Yaskawa INFORM job: R1_W01(KAMERA)(0,-90).JBI

/JOB
//NAME R1_W01(KAMERA)(0,-90)
//POS
///NPOS 10,10,0,0,0,0
///TOOL 0
///POSTYPE PULSE
///LIMIT ON
///PULSE
C00000=3343,-162524,-138229,-10688,931,-77458
C00001=3343,-162524,-138229,-10688,931,-77458
///LIMIT OFF
C00002=146555,-32624,-97126,-37706,85917,-68564
C00003=192498,68076,-33610,-32500,114040,-68788
C00004=185826,59216,-21978,-23322,112796,-65701
C00005=180860,70259,-8687,-21392,109491,-66464
C00006=183450,60909,-15972,-26835,103470,-66374
C00007=180988,72118,-8747,-21583,110442,-66611
C00008=181141,75755,-9105,-21978,112418,-66957
C00009=188486,40732,-78117,-36575,78939,-72193
BC00000=7717,939738,1042121
BC00001=7717,1361376,1042121
///LIMIT ON
BC00002=130580,1376610,1059176
BC00003=195745,1384690,1068222
BC00004=189788,1384690,1068222
BC00005=189788,1384690,1068222
BC00006=189789,1384690,1068220
BC00007=189953,1384690,1068222
BC00008=189837,1384690,1068222
BC00009=229747,1383410,1068222
//INST
///DATE 2024/07/30 12:51
///ATTR SC,RW
///GROUP1 RB1,BS1
NOP
'r1_W01(kamera)(0,-90)
'Path W401
SFTOF
MOVJ C00000 BC00000 VJ=100.00
MOVJ C00001 BC00001 VJ=100.00
MOVJ C00002 BC00002 VJ=100.00
MOVJ C00003 BC00003 VJ=70.00
MOVJ C00004 BC00004 VJ=20.00
MACRO1 MJ#(0) ARGF6
ARCON
MOVL C00005 BC00005 V=10.0
MOVL C00006 BC00006 V=10.0
ARCOF
MOVL C00007 BC00007 V=100.0
MOVL C00008 BC00008 V=166.7
MOVJ C00009 BC00009 VJ=100.00
END
